TYPE ST_CapPreScrewerParameters :
STRUCT
	lrTopZPosition						: LREAL;		//Pozycja bezpieczna załapywarki na osi pionowej
	lrPickZPosition						: LREAL;		//Wysokość pobierania
	lrPickYPosition						: LREAL;		//Pozycja osi poziomej do pobierania
	lrPlaceZPosition					: LREAL;		//Wysokość odkładania - koniec załapywania gwintu
	lrPlaceYPosition					: LREAL;		//Pozycja osi poziomej do odkładania
	lrCartesianCatchZPosition			: LREAL;		//Wysokość osi Z dla zamykania łapacza słomek
	lrCapCatcherZPosition				: LREAL;		//Wysokość zamykaniałapek zakrętek
	lrStrawCatcherZPosition				: LREAL;		//Wysokość otwierania łapaczy słomek
	LrCheckStrawCatcherActuatorZPosition: LREAL;		//
	lrScrewerStartZPosition				: LREAL;		//Wysokość początku zakręcania
	lrGripperOpenPosition				: LREAL;		//Wysokość otwierania chwytaka szyjki butelki
	lrCapCapCatcherRelese				: LREAL;		//Wysokość otwierania chwytaka nakrętki
	lrCatcherTopPosition				: LREAL;		//Pozycja górna osi łapaczy słomek
	lrCatcherCatchingPosition			: LREAL;		//Pozycja łapania słomki
	lrCatcherPlacePosition				: LREAL;		//Pozycja dolna łapacza słomki
	lrCatcherSpeed						: LREAL;		//Prędkość 
	lrCatcherAcceleration				: LREAL;		//Przyspieszenie 
	lrCatcherJerk						: LREAL;		//Zryw 
	lrPickerSpeed						: LREAL;		//Prędkość 
	lrPickerSpeedWhenScrewer			: LREAL;		//Prędkość osi Z przy zakręcaniu
	lrPickerAcceleration				: LREAL;		//Przyspieszenie 
	lrPickerJerk						: LREAL;		//Zryw 
	lrScrewDistance						: LREAL;		//Kąt zakręcania
	lrScrewFinding						: LREAL;		//Kąt szukania gwintu
	lrScrewSpeed						: LREAL;		//Prędkość zakręcania
	lrScrewAcceleration					: LREAL;		//Przyspieszenie
	lrScrewJerk							: LREAL;		//Zryw
	lrBendingDistance					: LREAL;		//Odległość zaokrąglania ruchów manipulatora
	lrStrawInsertDistance				: LREAL;		//Odległość wspulnego ruchu osi Z i łapacza słomek (prowadzenie słomki) 
	
	lrCatcherMaxHight					: LREAL;		//Wysokość maksymalan łapacza słomek
	lrCatcherMinHight					: LREAL;		//Wysokość minimalan łapacza słomek
	lrCatcherHightSV					: LREAL;		//Nastawa wysokości łapacza słomek
	rCatcherHightOffset					: REAL;			//Pozycja bazowania
	rPulseRatio							: REAL;			//
	
	bPickerActiv						: ARRAY [1..4] OF BOOL;
	tTimeVacuumWatchdog					: TIME;

	lrHeightAdditionalBlow				: LREAL;		//Wysokość aktywacji dodatkowego przedmuchu wszystkich ssawek (od zakończenia nakładania nasadki)
	
	//bPicker2Activ						: BOOL;
	//bPicker3Activ						: BOOL;
	//bPicker4Activ						: BOOL;
	
	tWaitInPlacePos						: TIME;
	
	bStrawCatcherON						: BOOL;			//Aktywacja pracy łapacza słomek
	bRejectON							: BOOL;			//Aktywacja odrzucania nasadek przy nieudanym pobraniu
	bVacuumDeactivate					: BOOL;			//Deaktywować podcisnienie
	
	sADS_NetId							: STRING;		//Adres net id dla komunikacji ADS
	nAxisY_ADS_SlaveAddr				: UINT;			//Adres urzadzenia dla komunikacji ADS
	nAxisZ_ADS_SlaveAddr				: UINT;			//Adres urzadzenia dla komunikacji ADS
	nCatcher_ADS_SlaveAddr				: UINT;			//Adres urzadzenia dla komunikacji ADS
	
	lrBottleHight						: LREAL;		//Wysokość butelki
	lrCapHight							: LREAL;		//Wysokość zamknięcia
	lrCapNeckHight						: LREAL;		//Wysokość szyjki zamknięcia
	
END_STRUCT
END_TYPE

(* stored: Version 1.2.0.0, ProductVersion 3.1.4026.13, FileIdentifier d87dd0ed0e55cbd912eb1bf01dd45ad796cb2451, FileSignature 6ffcbae4b60bbb48c53a0df5fb8e6cdec5e0f94138e643c915e6d0773b2b2aec459f7aa3780a7ec5c32209114b45a86d3bfd576b6b9a3718e3b28632358a1215331d07d2cc5a97bed6818209fdb87d8cd732c06aec575bb1f0f0b71f1c2411a7c28a855487dfa762a4b1c8ed5d5dcc59914695a38c86e65beb57f8c26be2041981a97e11fb6e91db7a607e00ec23532da82d10d4d065b6969e5d9b96aef991ed874028b94ebc397e6574bf5cce215607f742ca23c1f1c1492d48ceaefa1165c12d5d8b474e85157aa41ecbe1f35c06882cd17f47a8fb2ef37f8b8aea54abcee845ec58ab8dff335bfb02ab6d282d2e96726f4788cef4750ce39fad9e26644120
   DUT ST_CapPreScrewerParameters: Id {4dc5cd42-9fc9-4f4e-8ce5-45c7ad7a61fd} *)
